// TIA Portal V20 export
TYPE "LKinCtrl_PointEditor_typeHMIInterface"
// stored: Access Published
   STRUCT
      typeOfKinematics : DInt;
      interlockID : Int;
      pointTable : "LKinCtrl_PointEditor_typePointTable";
      pointConfiguration : "LKinCtrl_PointEditor_typePointConfiguration";
   END_STRUCT;
END_TYPE
